// Mitsubishi GX Works2 project: SKUBI_program_work_simplified   PLC: FX1N/FX1NC

PROGRAM MAIN
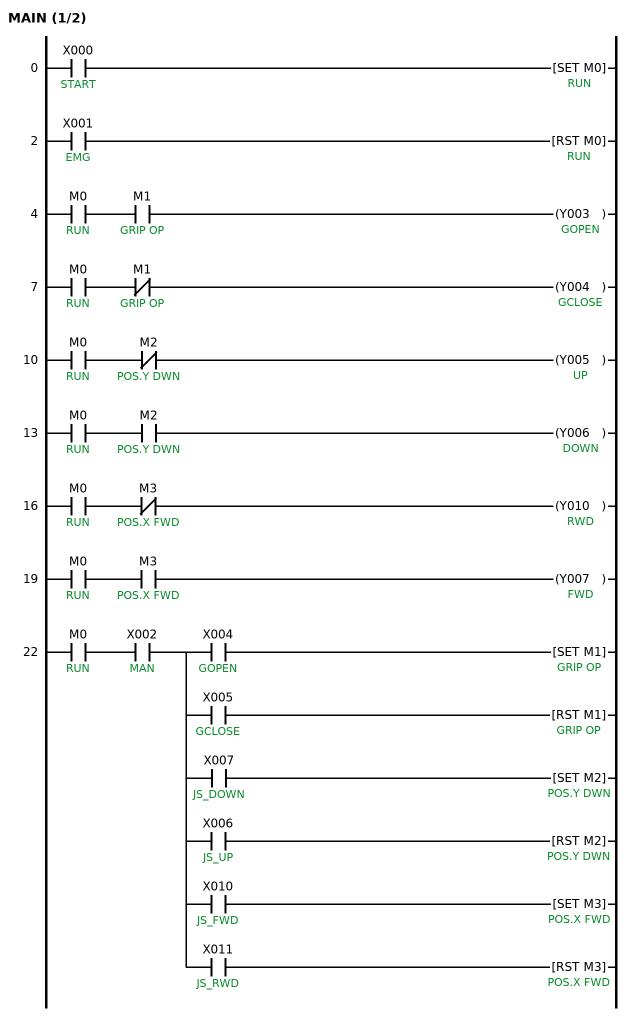
0     LD      X000  ; START
      SET     M0  ; RUN
2     LD      X001  ; EMG
      RST     M0  ; RUN
4     LD      M0  ; RUN
      AND     M1  ; GRIP OP
      OUT     Y003  ; GOPEN
7     LD      M0  ; RUN
      ANI     M1  ; GRIP OP
      OUT     Y004  ; GCLOSE
10    LD      M0  ; RUN
      ANI     M2  ; POS.Y DWN
      OUT     Y005  ; UP
13    LD      M0  ; RUN
      AND     M2  ; POS.Y DWN
      OUT     Y006  ; DOWN
16    LD      M0  ; RUN
      ANI     M3  ; POS.X FWD
      OUT     Y010  ; RWD
19    LD      M0  ; RUN
      AND     M3  ; POS.X FWD
      OUT     Y007  ; FWD
22    LD      M0  ; RUN
      AND     X002  ; MAN
      MPS
      AND     X004  ; GOPEN
      SET     M1  ; GRIP OP
      MRD
      AND     X005  ; GCLOSE
      RST     M1  ; GRIP OP
      MRD
      AND     X007  ; JS_DOWN
      SET     M2  ; POS.Y DWN
      MRD
      AND     X006  ; JS_UP
      RST     M2  ; POS.Y DWN
      MRD
      AND     X010  ; JS_FWD
      SET     M3  ; POS.X FWD
      MPP
      AND     X011  ; JS_RWD
      RST     M3  ; POS.X FWD
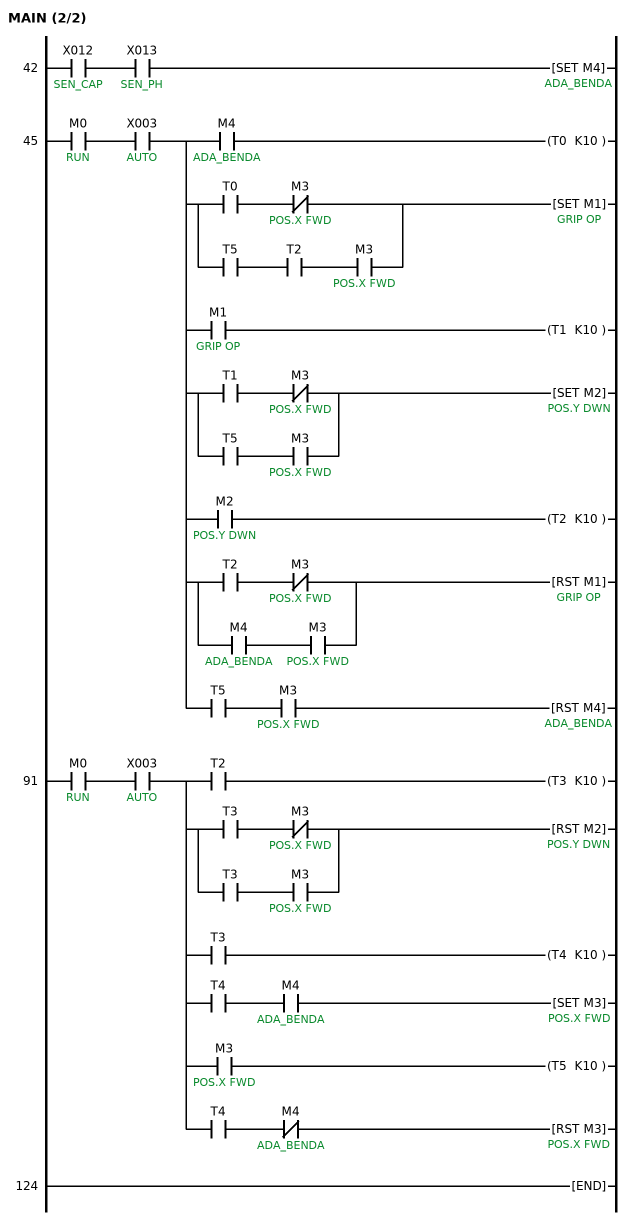
42    LD      X012  ; SEN_CAP
      AND     X013  ; SEN_PH
      SET     M4  ; ADA_BENDA
45    LD      M0  ; RUN
      AND     X003  ; AUTO
      MPS
      AND     M4  ; ADA_BENDA
      OUT     T0 K10
      MRD
      LD      T0
      ANI     M3  ; POS.X FWD
      LD      T5
      AND     T2
      AND     M3  ; POS.X FWD
      ORB
      ANB
      SET     M1  ; GRIP OP
      MRD
      AND     M1  ; GRIP OP
      OUT     T1 K10
      MRD
      LD      T1
      ANI     M3  ; POS.X FWD
      LD      T5
      AND     M3  ; POS.X FWD
      ORB
      ANB
      SET     M2  ; POS.Y DWN
      MRD
      AND     M2  ; POS.Y DWN
      OUT     T2 K10
      MRD
      LD      T2
      ANI     M3  ; POS.X FWD
      LD      M4  ; ADA_BENDA
      AND     M3  ; POS.X FWD
      ORB
      ANB
      RST     M1  ; GRIP OP
      MPP
      AND     T5
      AND     M3  ; POS.X FWD
      RST     M4  ; ADA_BENDA
91    LD      M0  ; RUN
      AND     X003  ; AUTO
      MPS
      AND     T2
      OUT     T3 K10
      MRD
      LD      T3
      ANI     M3  ; POS.X FWD
      LD      T3
      AND     M3  ; POS.X FWD
      ORB
      ANB
      RST     M2  ; POS.Y DWN
      MRD
      AND     T3
      OUT     T4 K10
      MRD
      AND     T4
      AND     M4  ; ADA_BENDA
      SET     M3  ; POS.X FWD
      MRD
      AND     M3  ; POS.X FWD
      OUT     T5 K10
      MPP
      AND     T4
      ANI     M4  ; ADA_BENDA
      RST     M3  ; POS.X FWD
124   END
END_PROGRAM
